// TIA Portal V20 export
DATA_BLOCK "ControlNodes"   // DB116
// stored: MemoryReserve 100, Namespace Unit1.Em5
   VAR
      em { ExternalWritable := 'False'} : "LAF_typeEmControlNode";
      cm { ExternalWritable := 'False'} : "Unit1.Em5.typeCmControlNode";
      citiMap : "LER_OEM_Data";
      ManualInput { ExternalWritable := 'False'} : "Unit1.Em5.typeSequenceControlNode";
   END_VAR
   VAR RETAIN
      cmNgAndManualInputAxisY { ExternalWritable := 'False'} : "LBC_typeAxis64PosControlNode";
      cmMagazineAxisZ { ExternalWritable := 'False'} : "LBC_typeAxis64PosControlNode";
      cmNgAndManualInputCylinderUpDown { ExternalWritable := 'False'} : "LBC_typeTwoWayActuatorControlNode";
      cmNgAndManualInputVacuum1OnOff { ExternalWritable := 'False'} : "LBC_typeTwoWayActuatorControlNode";
      cmNgAndManualInputVacuum2OnOff { ExternalWritable := 'False'} : "LBC_typeTwoWayActuatorControlNode";
      cmNgAndManualInputVibrator1OnOff { ExternalWritable := 'False'} : "LBC_typeTwoWayActuatorControlNode";
      cmNgAndManualInputVibrator2OnOff { ExternalWritable := 'False'} : "LBC_typeTwoWayActuatorControlNode";
      cmMagazineLockCylinderUpDown { ExternalWritable := 'False'} : "LBC_typeTwoWayActuatorControlNode";
      cmNgAndManaulInputMagazineElectrodeDetectionSensor { ExternalWritable := 'False'} : "LBC_typeDigitalSignalControlNode";
      cmNgAndManualInputMagazineDetectionSensor { ExternalWritable := 'False'} : "LBC_typeDigitalSignalControlNode";
      cmNgAndManualInputMagazineFullSensor { ExternalWritable := 'False'} : "LBC_typeDigitalSignalControlNode";
      cmNgAndManualInputElectrodeDetectionSensor { ExternalWritable := 'False'} : "LBC_typeDigitalSignalControlNode";
      cmMagazineSafetyPinIdlePosition { ExternalWritable := 'False'} : "LBC_typeDigitalSignalControlNode";
      cmNgAndManualInputAxisY_TorqueCal { ExternalWritable := 'False'} : "LER_typeServoTorqueCalControlNode";
      cmMagazineAxisZ_TorqueCal { ExternalWritable := 'False'} : "LER_typeServoTorqueCalControlNode";
   END_VAR
BEGIN
   // cm.brakeTest.magazine.monitoring.error : Magazine Axis Brake Test Error
   // cm.brakeTest.magazine.monitoring.busy : Magazine Axis Brake Test In progress
END_DATA_BLOCK
